FUNCTION_BLOCK WarpPolar (* openCV warp polar *)
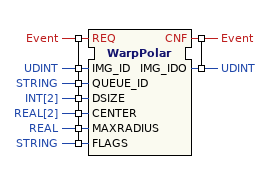
  EVENT_INPUT
    REQ WITH IMG_ID, QUEUE_ID, DSIZE, CENTER, MAXRADIUS, FLAGS;
  END_EVENT
  EVENT_OUTPUT
    CNF WITH IMG_IDO;
  END_EVENT
  VAR_INPUT
    IMG_ID : UDINT;
    QUEUE_ID : STRING;
    DSIZE : ARRAY [0..1] OF INT;
    CENTER : ARRAY [0..1] OF REAL;
    MAXRADIUS : REAL;
    FLAGS : STRING;
  END_VAR
  VAR_OUTPUT
    IMG_IDO : UDINT;
  END_VAR
END_FUNCTION_BLOCK
